// TIA Portal V20 export
VAR_GLOBAL   // PLC tag table "默认变量表"
   取芯V90_Actor_Interface_AddressIn AT %I82.0 : "PD_TEL3_IN";
   取芯V90_Actor_Interface_AddressOut AT %Q74.0 : "PD_TEL3_OUT";
   纠偏V90_Actor_Interface_AddressIn AT %I64.0 : "PD_TEL3_IN";
   纠偏V90_Actor_Interface_AddressOut AT %Q64.0 : "PD_TEL3_OUT";
   System_Byte AT %MB1 : Byte;
   FirstScan AT %M1.0 : Bool;
   DiagStatusUpdate AT %M1.1 : Bool;
   AlwaysTRUE AT %M1.2 : Bool;
   AlwaysFALSE AT %M1.3 : Bool;
   Clock_Byte AT %MB0 : Byte;
   Clock_10Hz AT %M0.0 : Bool;
   Clock_5Hz AT %M0.1 : Bool;
   "Clock_2.5Hz" AT %M0.2 : Bool;
   Clock_2Hz AT %M0.3 : Bool;
   "Clock_1.25Hz" AT %M0.4 : Bool;
   Clock_1Hz AT %M0.5 : Bool;
   "Clock_0.625Hz" AT %M0.6 : Bool;
   "Clock_0.5Hz" AT %M0.7 : Bool;
   纠偏V90控制字 AT %MW2 : Word;
   纠偏V90状态字 AT %MW4 : Word;
   纠_回原模式 AT %MW6 : Int;
   纠_绝对位置 AT %MD8 : Real;
   纠_相对位置 AT %MD12 : Real;
   纠_绝对速度 AT %MD16 : Real;
   纠_点动速度 AT %MD20 : Real;
   纠_当前位置 AT %M24.0 : LReal;
   纠_当前速度 AT %M32.0 : LReal;
   取芯V90控制字 AT %MW40 : Word;
   取芯V90状态字 AT %MW42 : Word;
   取_回原模式 AT %MW44 : Int;
   取_绝对位置 AT %MD46 : Real;
   取_绝对速度 AT %MD50 : Real;
   取_相对位置 AT %MD54 : Real;
   取_相对速度 AT %MD58 : Real;
   取_点动速度 AT %MD62 : Real;
   取_当前速度 AT %M66.0 : LReal;
   取_当前位置 AT %M74.0 : LReal;
END_VAR
